// TIA Portal project "Clase_con_ruben" (V15)

(* hardware
DEVICE "S7-1200 station_1"  S7-1200 Station
   slot 0: "Rack_0"  S7-1200 Rack  Rack  V1.0
   slot 1: "PLC_1"  CPU 1214C DC/DC/DC  6ES7 214-1AG40-0XB0  V4.2
*)

// ===== PLC "PLC_1"  CPU 1214C DC/DC/DC =====

VAR_GLOBAL   // PLC tag table "Tabla de variables estándar"
   "Clock_Byte" AT %MB500 : Byte;
   "Clock_10Hz" AT %M500.0 : Bool;
   "Clock_5Hz" AT %M500.1 : Bool;
   "Clock_2.5Hz" AT %M500.2 : Bool;
   "Clock_2Hz" AT %M500.3 : Bool;
   "Clock_1.25Hz" AT %M500.4 : Bool;
   "Clock_1Hz" AT %M500.5 : Bool;
   "Clock_0.625Hz" AT %M500.6 : Bool;
   "Clock_0.5Hz" AT %M500.7 : Bool;
   "segundos" AT %MW0 : Int;
   "FlancoPositivo" AT %M2.0 : Bool;
   "minutos" AT %MW4 : Int;
   "eventoup" AT %M2.1 : Bool;
   "eventodown" AT %M2.2 : Bool;
   "eventoreset" AT %M2.3 : Bool;
   "eventoLoad" AT %M2.4 : Bool;
   "salidaQu" AT %M2.5 : Bool;
   "salidaQd" AT %M2.6 : Bool;
   "SensordeNivel" AT %IW40 : Int;
   "normalizar" AT %MD6 : Real;
   "Altura0" AT %MD10 : Real;
   "Altura1" AT %MD14 : Real;
   "metrosH2o" AT %MD18 : Real;
END_VAR

// folder: System blocks/Program resources

DATA_BLOCK "IEC_Counter_0_DB_1"   // DB2
{ S7_Optimized_Access := 'TRUE' }
AUTHOR : Simatic
FAMILY : IEC
NAME : CNTR
VERSION : 1.0
// stored: InstanceOfName IEC_COUNTER
"IEC_COUNTER"
BEGIN
END_DATA_BLOCK

// folder: (top level)

ORGANIZATION_BLOCK "Main"   // OB1, LAD, ProgramCycle
TITLE = "Main Program Sweep (Cycle)"
{ S7_Optimized_Access := 'TRUE' }
VERSION : 0.1
   VAR_INPUT
      Initial_Call : Bool;   // Initial call of this OB
      Remanence : Bool;   // =True, if remanent data are available
   END_VAR
   VAR_TEMP   // added for the SCL form of the ladder/FBD networks
      _w1 : Bool;
   END_VAR
BEGIN

REGION Network 1
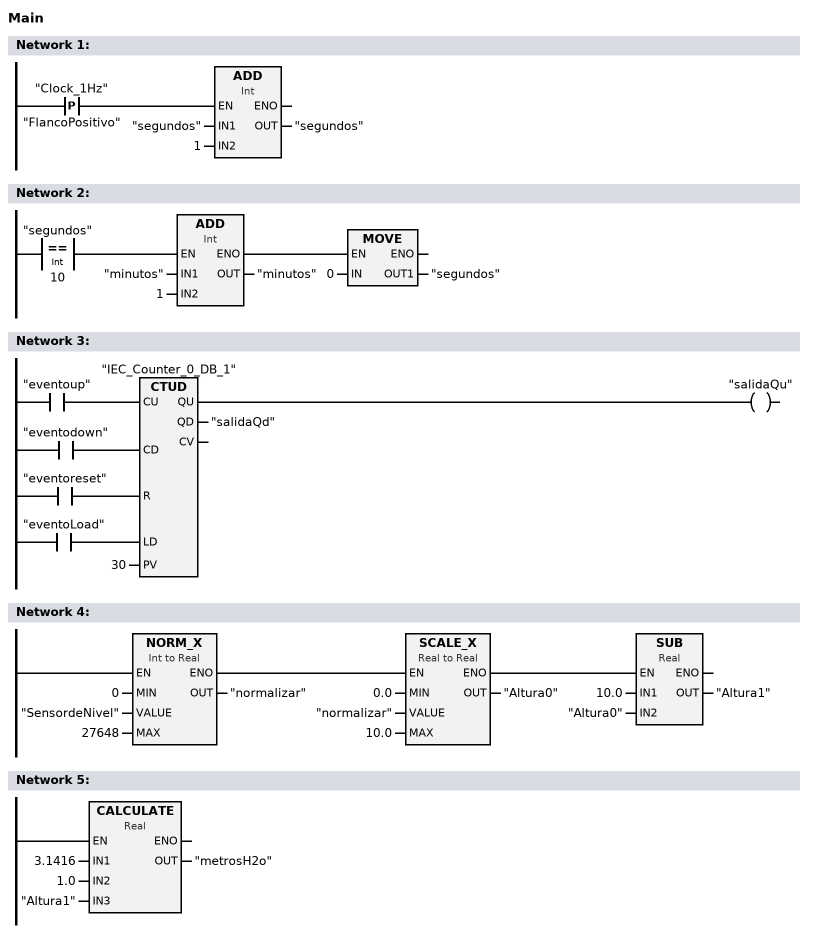
   RUNG wire#powerrail
      P_Contact(operand := "Clock_1Hz", bit := "FlancoPositivo")
      { S7_Templates := "SrcType := Int" } Add(in1 := "segundos", in2 := 1, out => "segundos")
   END_RUNG
   // the same network as SCL:
   #_w1 := "Clock_1Hz" AND NOT "FlancoPositivo";   // rising edge of "Clock_1Hz"
   "FlancoPositivo" := "Clock_1Hz";
   IF #_w1 THEN "segundos" := "segundos" + 1; END_IF;
END_REGION

REGION Network 2
   RUNG wire#powerrail
      { S7_Templates := "SrcType := Int" } EQ_Contact(in1 := "segundos", in2 := 10)
      { S7_Templates := "SrcType := Int" } Add(in1 := "minutos", in2 := 1, out => "minutos")
      Move(in := 0, out1 => "segundos")
   END_RUNG
   // the same network as SCL:
   IF "segundos" = 10 THEN
       "minutos" := "minutos" + 1;
       "segundos" := 0;
   END_IF;
END_REGION

REGION Network 3
   "IEC_Counter_0_DB_1".CTUD(CU := "eventoup",
                           CD := "eventodown",
                           R := "eventoreset",
                           LD := "eventoLoad",
                           PV := 30,
                           QD => "salidaQd");
   "salidaQu" := "IEC_Counter_0_DB_1".QU;
END_REGION

REGION Network 4
   RUNG wire#powerrail
      { S7_Templates := "[SrcType := Int, DestType := Real]" } Normalize(min := 0, value := "SensordeNivel", max := 27648, out => "normalizar")
      { S7_Templates := "[SrcType := Real, DestType := Real]" } Scale(min := 0.0, value := "normalizar", max := 10.0, out => "Altura0")
      { S7_Templates := "SrcType := Real" } Sub(in1 := 10.0, in2 := "Altura0", out => "Altura1")
   END_RUNG
   // the same network as SCL:
   "normalizar" := NORM_X(MIN := 0, VALUE := "SensordeNivel", MAX := 27648);
   "Altura0" := SCALE_X(MIN := 0.0, VALUE := "normalizar", MAX := 10.0);
   "Altura1" := 10.0 - "Altura0";
END_REGION

REGION Network 5
   RUNG wire#powerrail
      { S7_Templates := "SrcType := Real"; S7_Expression := "IN1*SQR(IN2)*IN3" } Calculate(in1 := 3.1416, in2 := 1.0, in3 := "Altura1", out => "metrosH2o")
   END_RUNG
   // the same network as SCL:
   "metrosH2o" := 3.1416*SQR(1.0)*"Altura1";
END_REGION
END_ORGANIZATION_BLOCK